FUNCTION CheckRangeSigned : DINT
VAR_INPUT
	value, lower, upper: DINT;
END_VAR

{noflow}

IF (value < lower) THEN
	CheckRangeSigned := lower;
	oaksGVL.udiCheckRangeSigned := oaksGVL.udiCheckRangeSigned + 1;
ELSIF(value > upper) THEN
	CheckRangeSigned := upper;
	oaksGVL.udiCheckRangeSigned := oaksGVL.udiCheckRangeSigned + 1;
ELSE
	CheckRangeSigned := value;
END_IF
{flow}

END_FUNCTION

(* stored: Version 1.1.0.1, ProductVersion 3.1.4022.18
   POU CheckRangeSigned: Id {cbb84e00-905b-4097-a7d7-2788f0873be9}, SpecialFunc CheckRangeSigned *)
